FUNCTION_BLOCK ConcreteAssertions EXTENDS CNM_AssertionInterfaceLib.AbstractAssertor IMPLEMENTS CNM_AssertionInterfaceTests.IAssertorContainer
VAR
	wrongAssertion	:BOOL;
END_VAR

METHOD assertionWasWrong
VAR_INPUT
	caller			:CNM_AbstractObject.IObject;
	message			:AssertMessage;
	additionalText	:Tc2_System.T_MaxString;
END_VAR
THIS^.wrongAssertion := TRUE;
END_METHOD

PROPERTY assertor : CNM_AssertionInterfaceTests.CNM_AssertionInterfaceLib.IAssertor
GET
assertor := THIS^;
END_GET
END_PROPERTY

PROPERTY className : CNM_AbstractObject.ClassName
GET
className := 'ConcreteAssertions';
END_GET
END_PROPERTY

METHOD resetAssertor
THIS^.wasAssertionWrong := FALSE;
END_METHOD

PROPERTY wasAssertionWrong : BOOL
GET
wasAssertionWrong := THIS^.wrongAssertion;
END_GET
SET
THIS^.wrongAssertion := wasAssertionWrong;
END_SET
END_PROPERTY

END_FUNCTION_BLOCK

(* stored: Version 1.1.0.1, ProductVersion 3.1.4024.12
   POU ConcreteAssertions: Id {81987a0e-d932-45b6-ab4b-b2c6b593d05f}, SpecialFunc None
   Method assertionWasWrong: Id {86beb84b-11a1-4994-8a22-1223b2108d6e}
   Property assertor: Id {a62cdb6e-56fd-4462-a276-71e81161234c}
   Get Get: Id {9f4ac83f-a96b-44f1-b934-b437662da28e}
   Property className: Id {31a7334d-7454-4b79-9894-5185decc6e93}
   Get Get: Id {a2ef7755-faad-44dd-b625-8a084e287aff}
   Method resetAssertor: Id {60871598-b112-4277-8f57-07b9c429874b}
   Property wasAssertionWrong: Id {d15b8142-368c-4004-93b7-a6615ae61805}
   Get Get: Id {4134aee8-9d1f-4c1b-a289-44894e17f9b3}
   Set Set: Id {f1235e34-ffc0-4fce-aac4-366234334135} *)
